FUNCTION_BLOCK FINAL ExtendedLoggerEnrichmentConfiguration EXTENDS TcoLoggerEnrichmentConfiguration
VAR_INPUT
END_VAR
VAR_OUTPUT
END_VAR
VAR
	_projectNameEnricher		: ProjectNameEnricher;
END_VAR

METHOD PUBLIC ProjectName : REFERENCE TO TcoLoggerConfiguration
VAR_INPUT
END_VAR
_config.AddEnrichment(_projectNameEnricher);
ProjectName := _config;
END_METHOD

END_FUNCTION_BLOCK

(* stored: Version 1.1.0.1, ProductVersion 3.1.4024.9
   POU ExtendedLoggerEnrichmentConfiguration: Id {846196e7-d5f8-0d92-0d5a-197d23edf8ac}, SpecialFunc None
   Method ProjectName: Id {4c001959-9514-0eca-33f0-11636b75be71} *)
